FUNCTION TryConvert_UINT_TO_LINT : BOOL
VAR_INPUT
	in : UINT;
	out : REFERENCE TO LINT;
END_VAR

out := UINT_TO_LINT(in);
TryConvert_UINT_TO_LINT := TRUE;

END_FUNCTION

(* stored: Version 1.1.0.1, ProductVersion 3.1.4024.12
   POU TryConvert_UINT_TO_LINT: Id {6a0b8821-9acd-4422-8bd7-754cb3c254b9}, SpecialFunc None *)
